TYPE CmpConvBreakStopGroupConfig :
STRUCT
	NumberStops : DINT;
	BreakStopDefault: BreakStopConfig;
	BreakStops: ARRAY[1..cBreakStopGroupMaxInstance] OF BreakStopConfig;
END_STRUCT
END_TYPE

(* stored: Version 1.1.0.1, ProductVersion 3.1.4024.6
   DUT CmpConvBreakStopGroupConfig: Id {ad750131-a14e-4534-afcc-88aeed92580f} *)
